Yaskawa INFORM job: TESTKAMERA.JBI

/JOB
//NAME TESTKAMERA
//POS
///NPOS 7,7,0,0,0,0
///TOOL 0
///POSTYPE PULSE
///PULSE
C00000=115133,-18045,-5914,51808,64300,77694
C00001=119045,12059,21912,51887,61054,77964
C00002=119045,12059,21912,51887,61054,77964
C00003=119210,35382,44396,52673,59799,77242
C00004=119389,77682,92841,56818,54888,73750
C00005=118037,44157,51798,52848,60437,76945
C00006=115704,40745,42367,51543,64300,78025
BC00000=388872,392350,408016
BC00001=388872,392350,408016
BC00002=388872,392350,408016
BC00003=388872,392350,408016
BC00004=388872,392350,408016
BC00005=388872,392350,408016
BC00006=388872,392350,408016
//INST
///DATE 2023/11/02 15:04
///ATTR SC,RW
///GROUP1 RB1,BS1
///LVARS 0,0,0,0,0,0,0,0
NOP
SFTOF
'-- TL mode [B000]-------------
'- 0:NO TRACKING, 1:TRACKING --
'------------------------------
SET B000 1
MOVJ C00000 BC00000 VJ=5.00
MACRO1 MJ#(5) ARGFB000 ARGF1 ARGF80 ARGFC00001 ARGFBC00001 ARGF7
MOVL C00002 BC00002 V=13.3
'arcon
MOVL C00003 BC00003 V=13.3
MACRO1 MJ#(9) ARGFB000 ARGF1
MOVL C00004 BC00004 V=13.3
'arcof
MACRO1 MJ#(3) ARGFB000
MOVL C00005 BC00005 V=16.7
MOVJ C00006 BC00006 VJ=5.00
END
